(* PLC project Untitled1, Beckhoff Automation GmbH TwinCAT PLC Control 3.5.13.21 *)
(* stored: creationDateTime 2022-05-13T11:55:24.4715014, modificationDateTime 2022-05-13T11:55:24.4715014 *)

VAR_GLOBAL  (* GVL_AutoGenerated *)
  EtherCATStatus AT %Q* : UINT;
  EtherCAT_CoEWriteExecute AT %I* : BOOL;
  EtherCAT_CoEWriteError AT %Q* : BOOL;
  EtherCAT_CoEWriteDone AT %Q* : BOOL;
  EtherCAT_CoEWriteSlaveAddr AT %I* : UINT;
  EtherCAT_CoEWriteIndex AT %I* : WORD;
  EtherCAT_CoEWriteSubIndex AT %I* : BYTE;
  EtherCAT_NetId AT %I* : AMSNETID;
  EtherCATChangeCount AT %Q* : ARRAY[1..50] OF UINT;
  EtherCATChangeCountReset AT %I* : BOOL;
END_VAR
